Staubli VAL3: Motion.dtx

bool bIsScara = true
bool bLinear = true
bool bLizOK = true
bool bReset
bool bSkipVersionChk
bool bStopAll
bool bThruDwnEnabled
bool bThruUpEnabled
dio doThruDwnLimit
dio doThruUpLimit
frame fConveyor = {x=650.958732, y=458.882506, z=-86.396059, rx=0.033285, ry=0.199699, rz=-179.551413, fatherId=world[0]}
frame fMobileFrame[10]
  [0] = {x=3129.225307, fatherId=fConveyor[0]}
  [1] = {x=3129.220405, fatherId=fConveyor[0]}
  [2] = {x=3129.171164, fatherId=fConveyor[0]}
  [3] = {fatherId=fConveyor[0]}
  [4] = {fatherId=fConveyor[0]}
  [5] = {fatherId=fConveyor[0]}
  [6] = {fatherId=fConveyor[0]}
  [7] = {fatherId=fConveyor[0]}
  [8] = {fatherId=fConveyor[0]}
  [9] = {fatherId=fConveyor[0]}
mdesc mTrackOff = {accel=25, vel=50, decel=25, blend=cartesian, leave=20, reach=20}
mdesc mTrackOn = {accel=169, vel=130, decel=169, blend=cartesian, leave=20, reach=20}
mdesc mTracking
num nCnvSynch
num nConveyorSpeed = 518.670703
num nDEFAULTTRKZONE = -99
num nIdxID
num nIdxStatus
num nLinkedTo[10]
  [3] = -1
  [4] = -1
  [5] = -1
  [6] = -1
  [7] = -1
  [8] = -1
  [9] = -1
num nMAXMOBILEFRAME = 10
num nMobFrameSync = -1
num nPosInQueue[10]
  [0] = 2
  [1] = 2
  [2] = 2
  [3] = -1
  [4] = -1
  [5] = -1
  [6] = -1
  [7] = -1
  [8] = -1
  [9] = -1
num nStatus
num nTrackZonPrev = -99
num nTrackingZone = -99
pointRs pInterTrack_RS = {fatherId=fMobileFrame[0]}
pointRs pTrackOff_RS = {x=-127.749433, y=517.878584, z=103.849179, rx=-179.965152, ry=-0.199433, rz=0.448706, shoulder=lefty, fatherId=fConveyor[0]}
pointRs pTrackOn_RS = {x=72.083546, y=72.428021, z=77.085378, rx=-0.209053, ry=-179.916469, rz=-18.008681, shoulder=righty, fatherId=fMobileFrame[2]}
pointRs pTracking_RS = {fatherId=fMobileFrame[0]}
pointRx pInterTrack = {fatherId=fMobileFrame[0]}
pointRx pTrackOff = {fatherId=fConveyor[0]}
pointRx pTrackOn = {fatherId=fMobileFrame[0]}
pointRx pTracking = {fatherId=fMobileFrame[0]}
string sConveyorList = "cvIn"
string sErrMsgList[20]
  [0] = "Not initialized"
  [1] = "Running. No tracking move command pending."
  [2] = "Internal run-time error in task called *\../*. Error code is *. Refer to valTrack Reference guide for more details"
  [3] = "The tracking is in error"
  [4] = "A trackOn command is being executed."
  [5] = "A tracking move command (linear or circular) is being executed."
  [6] = "The arm is tracking a fixed point on a conveyor."
  [9] = "Warning, the add on called "expansion" is required with this VAL3 version"
  [11] = "Warning, libraries for conveyor tracking require VAL3 version s7.6.0 or higher"
  [12] = "MOT>>Number of conveyor is limited to *"
  [13] = "MOT>>The library *\../* used as conveyor number * was not loaded because of error code *"
  [14] = "MOT(init)>>Cannot convert frame number * to mobile frame"
string sErrorMessage = "Running. No tracking move command pending."
string sTASK = "tracking"
tool tTool = {x=-8.16, y=18.26, z=80, rz=110, fatherId=flange[0], ioLink=valve1}
